FUNCTION_BLOCK T_MockTask IMPLEMENTS I_Task
VAR_INPUT
  _busy : BOOL;
  _done : BOOL;
  _error : BOOL;
END_VAR
VAR
  state, prevState : (IDLE_STATE, BUSY_STATE, DONE_STATE, ERROR_STATE);
  counter : UINT := 0;
  cycleCount : UINT := 0;
END_VAR

METHOD Abort
// no op
END_METHOD

{warning 'add property implementation'}
PROPERTY Available : BOOL
GET
END_GET
END_PROPERTY

PROPERTY Busy : BOOL
GET
Busy := _busy;
END_GET
END_PROPERTY

METHOD PUBLIC CauseError
state := ERROR_STATE;
END_METHOD

METHOD PUBLIC CyclicLogic
CASE state OF
  IDLE_STATE:
    IF StateChanged() THEN
      _Busy := FALSE;
      _Done := FALSE;
      _Error := FALSE;
    END_IF
    
  BUSY_STATE:
    IF StateChanged() THEN
      _Busy := TRUE;
      _Done := FALSE;
      _Error := FALSE;
    END_IF

    IF NOT WaitForCycles(cycleCount) THEN
      RETURN;
    END_IF

    state := DONE_STATE;

  DONE_STATE:
    IF StateChanged() THEN
      _Busy := FALSE;
      _Done := TRUE;
      _Error := FALSE;
    END_IF

  ERROR_STATE:
    IF StateChanged() THEN
      _Error := TRUE;
      _Busy := FALSE;
      _Done := FALSE;
    END_IF

END_CASE
END_METHOD

PROPERTY Done : BOOL
GET
Done := _done;
END_GET
END_PROPERTY

METHOD PUBLIC DoSomething : I_Task
VAR_INPUT
  busyCycles : UINT;
END_VAR
state := BUSY_STATE;
cycleCount := busyCycles;
DoSomething := THIS^;
END_METHOD

PROPERTY Error : BOOL
GET
Error := _error;
END_GET
END_PROPERTY

{warning 'add property implementation'}
PROPERTY ErrorId : STRING
GET
END_GET
END_PROPERTY

METHOD Execute : BOOL
// no ops
END_METHOD

{warning 'add method implementation '}
METHOD Free
END_METHOD

METHOD PRIVATE StateChanged : BOOL
IF  state = prevState THEN
  RETURN;
END_IF

prevState := state;
StateChanged := TRUE;
END_METHOD

{warning 'add property implementation'}
PROPERTY Timeout : BOOL
GET
END_GET
END_PROPERTY

METHOD PRIVATE WaitForCycles : BOOL
VAR_INPUT
  maxCount : UINT;
END_VAR
counter := counter + 1;

IF counter = maxCount THEN
  counter := 0;
  WaitForCycles := TRUE;
END_IF
END_METHOD

END_FUNCTION_BLOCK

(* stored: Version 1.1.0.1, ProductVersion 3.1.4024.12
   POU T_MockTask: Id {43a05129-dd0e-4806-bc27-45cfa44f475a}, SpecialFunc None
   Method Abort: Id {aeaaf20e-1dba-4044-a2a5-a6790b75bb15}
   Property Available: Id {68f0a419-ef81-4d1d-8746-fd1c7edec15a}
   Get Get: Id {5614d75b-9a84-4002-95b7-421e16d8a277}
   Property Busy: Id {14358a0e-f9ec-4a61-8586-1bb908feca6f}
   Get Get: Id {25afbc35-26ad-419f-8cfd-d6944eab2a89}
   Method CauseError: Id {426cbcf7-5f78-4956-a3bd-ae341fa1054a}
   Method CyclicLogic: Id {08e12be7-fac3-4c20-aa7e-4323956f8553}
   Property Done: Id {58c7844b-ed72-44bf-88a9-7f91052c7931}
   Get Get: Id {01b0135c-7796-4213-b5b0-69a041d02f51}
   Method DoSomething: Id {801f9f38-d8ce-4ba0-9d6e-b5e47aceffec}
   Property Error: Id {007f92b7-0637-4039-8ff8-aac93fabbd50}
   Get Get: Id {2d2574a8-79df-4e54-bb49-cc07d48f9e90}
   Property ErrorId: Id {8cf4a52d-3206-4ea8-b2f7-fae176174b25}
   Get Get: Id {79016913-a789-4cb7-ade6-1968b45dc697}
   Method Execute: Id {dd8509dd-9503-4514-a63c-450341e033ce}
   Method Free: Id {80c9c330-88a7-4772-9cdb-f4e5b430648b}
   Method StateChanged: Id {c26c9b0f-b443-4f87-827f-ae41025c6cbe}
   Property Timeout: Id {243e1fde-411e-4bcf-919a-f4825bc10afe}
   Get Get: Id {85347383-eb06-4d7e-9118-62b21cc22010}
   Method WaitForCycles: Id {ab9c58c6-8236-4eb0-b571-4567a7f2f18a} *)
